FUNCTION_BLOCK F_WSTRING_TO_DINT (* convert WSTRING to DINT *)
  (* Standard: 61131-3; Classification: type conversion function *)
  (* Version 0.0, 2013-08-29, 4DIAC-IDE, 4DIAC-Consortium *)
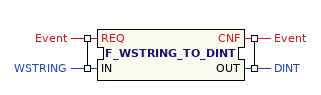
  EVENT_INPUT
    REQ WITH IN; (* Service Request *)
  END_EVENT
  EVENT_OUTPUT
    CNF WITH OUT; (* Confirmation of Requested Service *)
  END_EVENT
  VAR_INPUT
    IN : WSTRING; (* Event Input Qualifier *)
  END_VAR
  VAR_OUTPUT
    OUT : DINT; (* Event Output Qualifier *)
  END_VAR
END_FUNCTION_BLOCK
